TYPE WcState :
STRUCT
    State AT %I* : BOOL;
    InputToggle AT %I* : BOOL;
END_STRUCT
END_TYPE

(* stored: Version 1.1.0.1, ProductVersion 3.1.4024.9
   DUT WcState: Id {17cec864-319a-0250-26fc-c565083022ba} *)
